TYPE DUT_1 :
STRUCT
END_STRUCT
END_TYPE

(* stored: Version 1.1.0.1, ProductVersion 3.1.4024.13
   DUT DUT_1: Id {d23f96d3-6601-42a0-b830-ac4a515bff06} *)
